{attribute 'qualified_only'}
{attribute 'strict'}
TYPE E_DeliveryStatus :
(
	eNO_DELIVERY_INFORMATION := 0,
	eDELIVERY_OK,
	eDELIVERY_REJECTED
)UINT;
END_TYPE

(* stored: Version 1.1.0.1, ProductVersion 3.1.4022.12
   DUT E_DeliveryStatus: Id {95188abe-cae3-4846-862f-00d85e739980} *)
